FUNCTION F_CmpTimeSchedule : BOOL
VAR_INPUT
	timeToActivate:stTimeToSchedule2;	(*Hora para ligar a saida*)
	timeToDeactivate:stTimeToSchedule2;	(*Hora para desligar a saida*)
END_VAR
VAR
END_VAR

F_CmpTimeSchedule:=(timeToDeactivate.wHour>timeToActivate.wHour) OR ((timeToDeactivate.wHour = timeToActivate.wHour) AND (timeToDeactivate.wMinute> timeToActivate.wMinute));

END_FUNCTION

(* stored: Version 1.1.0.1, ProductVersion 3.1.4020.6
   POU F_CmpTimeSchedule: Id {c7799ba5-419f-4f2c-b1c8-7626f51be361}, SpecialFunc None *)
